FUNCTION_BLOCK FB_RunningState IMPLEMENTS I_State
VAR_INPUT
END_VAR
VAR_OUTPUT
END_VAR
VAR
	pConveyorSystem : POINTER TO FB_ConveyorSystem;
END_VAR

{warning 'add property implementation'}
PROPERTY Description : STRING
GET
Description := 'Running state';
END_GET
END_PROPERTY

{warning 'add method implementation '}
METHOD DetectedPartSensor1 : BOOL
END_METHOD

{warning 'add method implementation '}
METHOD DetectedPartSensor2 : BOOL
pConveyorSystem^.SetState(pConveyorSystem^.IdleState);
END_METHOD

{warning 'add method implementation '}
METHOD DetectedWeightSensor : BOOL
VAR
	fWeight : REAL;
	fbRandomNumber : DRAND;
END_VAR
IF pConveyorSystem^.aItemWeights[pConveyorSystem^.nCount] = 0 THEN
	pConveyorSystem^.SetState(pConveyorSystem^.IdleState);
	fbRandomNumber(SEED := 1, Num => fWeight);
	fWeight := fWeight * 1000 + 5.0;
	pConveyorSystem^.SetWeight(fWeight);
END_IF
END_METHOD

METHOD FB_init : BOOL
VAR_INPUT
	bInitRetains : BOOL; // if TRUE, the retain variables are initialized (warm start / cold start)
	bInCopyCode : BOOL;  // if TRUE, the instance afterwards gets moved into the copy code (online change)
	pConveyorSystem : POINTER TO FB_ConveyorSystem;
END_VAR
THIS^.pConveyorSystem := pConveyorSystem;
END_METHOD

{warning 'add method implementation '}
METHOD PressEmergencyStop : BOOL
pConveyorSystem^.SetState(pConveyorSystem^.EmergencyStopState);
END_METHOD

{warning 'add method implementation '}
METHOD PressStart : BOOL
END_METHOD

{warning 'add method implementation '}
METHOD PressStop : BOOL
END_METHOD

{warning 'add method implementation '}
METHOD ProcessedWeight : BOOL
END_METHOD

END_FUNCTION_BLOCK

(* stored: Version 1.1.0.1, ProductVersion 3.1.4024.12
   POU FB_RunningState: Id {5ced025a-cdbb-4bfd-aed6-e63f3e04df8b}, SpecialFunc None
   Property Description: Id {483a0495-1b7c-4bd5-8b39-3853b34c992a}
   Get Get: Id {3bb49784-7f07-44db-8ce1-d6b429b4a209}
   Method DetectedPartSensor1: Id {b6e721e9-1198-412b-8ade-e1726be0b72f}
   Method DetectedPartSensor2: Id {a8d2e503-f120-4838-9be8-38869cca7b99}
   Method DetectedWeightSensor: Id {ade77ac5-e2fc-4cfb-8cb0-1c03c6c27c99}
   Method FB_init: Id {ee0d9f84-997e-4011-9258-fb3236e92f84}
   Method PressEmergencyStop: Id {c867ca6c-f8c8-4393-ab87-257387785204}
   Method PressStart: Id {e3d979a2-19ab-4e98-abf7-24f0591f8b6f}
   Method PressStop: Id {0b53e972-ca65-43a9-a88a-47ea55764d9f}
   Method ProcessedWeight: Id {b219b61f-c763-492c-aa85-e029902ce541} *)
